INTERFACE I_INFLUXDB_ADS EXTENDS I_GENERAL_OBJECT

METHOD M_BucketExistCheck : BOOL
VAR_INPUT
  /// Name of the table that is to be read.
  sBucketName:                T_MaxString;
END_VAR
VAR_OUTPUT
  /// Result
  bResult:                    BOOL;
END_VAR
END_METHOD

METHOD M_ClearMeasurement : BOOL
VAR_INPUT
  /// Bucket name
  sBucketName:          T_MaxString;
  /// Name of the measure to clear
  sMeasurementName:     T_MaxString;
  /// From date time (Range)
  dtFrom:               DT;
  /// To date time (Range)
  dtTo:                 DT;
END_VAR
VAR_OUTPUT
	/// Result
	bResult	: BOOL;
END_VAR
END_METHOD

METHOD M_DeleteAllMeasurements : BOOL
VAR_INPUT
  /// Bucket name
  sBucketName:          T_MaxString;
END_VAR
VAR_OUTPUT
	/// Result
	bResult	: BOOL;
END_VAR
END_METHOD

METHOD M_DeleteField : BOOL
VAR_INPUT
  /// Bucket name
  sBucketName:          T_MaxString;
  /// Measurement Name
  sMeasurementName:     T_MaxString;
  /// Tag Name
  sTagName:             T_MaxString;
  /// Field Name
  sFieldName:           T_MaxString;
END_VAR
VAR_OUTPUT
  /// Result
  bResult:              BOOL;
END_VAR
END_METHOD

METHOD M_DeleteMeasurement : BOOL
VAR_INPUT
  /// Bucket name
  sBucketName:          T_MaxString;
  /// Name of the measure to delete.
  sMeasurementName:     T_MaxString;
END_VAR
VAR_OUTPUT
	/// Result
	bResult	: BOOL;
END_VAR
END_METHOD

METHOD M_DeleteTag : BOOL
VAR_INPUT
  /// Bucket name
  sBucketName:          T_MaxString;
  /// Measurement Name
  sMeasurementName:     T_MaxString;
  /// Tag Name
  sTagName:             T_MaxString;
END_VAR
VAR_OUTPUT
  /// Result
  bResult:              BOOL;
END_VAR
END_METHOD

METHOD M_DeleteTagContentBlock : BOOL
VAR_INPUT
  /// Bucket name
  sBucketName:          T_MaxString;
  /// Measurement Name
  sMeasurementName:     T_MaxString;
  /// Tag Name
  sTagName:             T_MaxString;
  /// Date and time from
  dtFrom:               DT;
  /// Date and Time to
  dtTo:                 DT;
END_VAR
VAR_OUTPUT
  /// Result
  bResult:              BOOL;
END_VAR
END_METHOD

METHOD M_FieldExistCheck : BOOL
VAR_INPUT
  /// Bucket name
  sBucketName:          T_MaxString;
  /// Measurement Name
  sMeasurementName:     T_MaxString;
  /// Tag Name
  sTagName:             T_MaxString;
  /// Field Name
  sFieldName:           T_MaxString;
END_VAR
VAR_OUTPUT
  /// Result
  bResult:              BOOL;
END_VAR
END_METHOD

METHOD M_GetTotalMeasurements : BOOL
VAR_INPUT
  /// Bucket name
  sBucketName:          T_MaxString;
END_VAR
VAR_OUTPUT
  /// Process success
  bResult:              BOOL;
  /// Result value
  uiResult:             UINT;
END_VAR
END_METHOD

METHOD M_MeasurementExistCheck : BOOL
VAR_INPUT
  /// Bucket name
  sBucketName:          T_MaxString;
  /// Name of the table that is to be read.
  sMeasurementName:     T_MaxString;
END_VAR
VAR_OUTPUT
  /// Result
  bResult:              BOOL;
END_VAR
END_METHOD

METHOD M_Reset : BOOL
VAR_INPUT
END_VAR
END_METHOD

METHOD M_SetReady : BOOL
VAR_INPUT
END_VAR
END_METHOD

METHOD M_TagExistCheck : BOOL
VAR_INPUT
  /// Bucket name
  sBucketName:          T_MaxString;
  /// Measurement Name
  sMeasurementName:     T_MaxString;
  /// Tag Name
  sTagName:             T_MaxString;
END_VAR
VAR_OUTPUT
  /// Result
  bResult:              BOOL;
END_VAR
END_METHOD

METHOD M_WriteStruct : BOOL
VAR_INPUT
  /// Bucket name
	sBucketName:                  T_MaxString;
	/// Name of the table that is to be read.
	sMeasurementName:             T_MaxString;
	/// Tag name
	sTagName:                     T_MaxString;
  /// Field values list
	stFieldValues:                ST_DATABASE_RECORD;
  /// Field struct content (Variable names)
  //pFieldStructContent:        POINTER TO ARRAY [0..99] OF T_MaxString;
	/// Field names list: names that appear in the database
	//pFieldNames:                POINTER TO ARRAY [0..99] OF T_MaxString;
END_VAR
VAR_OUTPUT
	/// Result
	bResult	: BOOL;
END_VAR
END_METHOD

PROPERTY P_ADSLifeBit : BOOL
GET
END_GET
END_PROPERTY

PROPERTY P_ADSState : BOOL
GET
END_GET
END_PROPERTY

PROPERTY P_Connected : BOOL
GET
END_GET
END_PROPERTY

PROPERTY P_Error : BOOL
GET
END_GET
END_PROPERTY

PROPERTY P_InfluxDBLifeBit : BOOL
GET
END_GET
END_PROPERTY

PROPERTY P_InfluxDBState : BOOL
GET
END_GET
END_PROPERTY

END_INTERFACE

(* stored: Version 1.1.0.1, ProductVersion 3.1.4024.12
   Itf I_INFLUXDB_ADS: Id {36104397-a43f-4b81-b638-271868415494}
   Method M_BucketExistCheck: Id {d0fa881f-3de0-4c5a-8233-22e7dc743627}
   Method M_ClearMeasurement: Id {dc135dc0-c001-48a7-a86a-9add3729f568}
   Method M_DeleteAllMeasurements: Id {f2dc2a94-b9e8-4b34-8895-4dbc6fe39456}
   Method M_DeleteField: Id {0ecbf110-a404-4085-9681-c0c2596ad7ab}
   Method M_DeleteMeasurement: Id {c1b7daa6-4e94-43c6-9dd1-3b33e13c06da}
   Method M_DeleteTag: Id {eeb750fe-0780-4ad6-8029-ad5c8f489a2b}
   Method M_DeleteTagContentBlock: Id {cee02e52-e90c-4c11-9a56-05be34f32760}
   Method M_FieldExistCheck: Id {788a0671-6798-4f19-a721-950e7abec066}
   Method M_GetTotalMeasurements: Id {98acedfa-acd6-4ef2-baea-997804b80257}
   Method M_MeasurementExistCheck: Id {6bcb11f7-77bd-4d3b-9d3d-74f084faf46c}
   Method M_Reset: Id {59c2e65f-e4aa-4f14-9820-a6d87d890064}
   Method M_SetReady: Id {48e70524-8888-4774-8246-dc992dda1d28}
   Method M_TagExistCheck: Id {77be6f17-e11f-4c2c-a323-95e172763d09}
   Method M_WriteStruct: Id {8e259580-aad4-4463-ba27-cb8cf68a3c7a}
   Property P_ADSLifeBit: Id {45014879-71dd-49ed-8686-2c335d4d29d2}
   Get Get: Id {6af7a5fa-5458-4df5-9561-1da6f35bd531}
   Property P_ADSState: Id {ed9b6413-4f61-4045-b0ce-2bdf6ddef539}
   Get Get: Id {368473b7-d912-489d-bbe6-b080809e86bb}
   Property P_Connected: Id {bb335fe8-81c2-467f-ba49-82e913a6c96c}
   Get Get: Id {b404539a-8b5c-4587-b77a-23449b126251}
   Property P_Error: Id {82258349-f26f-450c-a51f-732909dddf4e}
   Get Get: Id {88add42a-6233-42a5-a7b2-0b5718793b8e}
   Property P_InfluxDBLifeBit: Id {917d3f54-babb-4154-b8ad-57d8f4d1db23}
   Get Get: Id {7c183ad5-35c8-46eb-98c6-25c8406720ae}
   Property P_InfluxDBState: Id {e7d31142-16a8-4414-80a0-5ac8ca156b07}
   Get Get: Id {5089df90-ceac-43eb-b0fc-f496e81b0499} *)
